FUNCTION VelocitySaturation : LREAL
VAR_IN_OUT
	velocity : LREAL;
	max_velocity : LREAL;
	min_velocity : LREAL;
END_VAR

IF velocity > max_velocity THEN
	velocity := max_velocity;
END_IF
IF velocity < min_velocity THEN
	velocity := min_velocity;
END_IF

END_FUNCTION

(* stored: Version 1.1.0.1, ProductVersion 3.1.4024.11
   POU VelocitySaturation: Id {cdf42157-1b62-4c84-b11b-9950500958e8}, SpecialFunc None *)
